// TIA Portal project "Street Light Control" (V17)
// Street Light Control
// The Street Light gets ON for 20s when there is any movement detected and then blinks with a interval of 1s, gets turned OFF after 30s.

(* hardware
DEVICE "S7-1200 station_1"  S7-1200 Station
   slot 0: "Rack_0"  S7-1200 Rack  Rack  V1.0
   slot 1: "PLC_1"  CPU 1215C DC/DC/DC  6ES7 215-1AG40-0XB0  V4.5
*)

// ===== PLC "PLC_1"  CPU 1215C DC/DC/DC =====

VAR_GLOBAL   // PLC tag table "Default tag table"
   "Motion_Sensor" AT %I0.1 : Bool;
   "Street_Lights" AT %Q0.0 : Bool;
   "Tag_1" AT %M0.0 : Bool;
   "Tag_2" AT %M0.1 : Bool;
   "Tag_3" AT %MD0 : Time;
   "Tag_4" AT %MD4 : Time;
   "PB" AT %I0.0 : Bool;
   "Tag_5" AT %M0.3 : Bool;
END_VAR

// folder: System blocks/Program resources

DATA_BLOCK "IEC_Timer_0_DB"   // DB1
{ S7_Optimized_Access := 'TRUE' }
AUTHOR : Simatic
FAMILY : IEC
NAME : IEC_TMR
VERSION : 1.0
// stored: InstanceOfName IEC_TIMER
"IEC_TIMER"
BEGIN
END_DATA_BLOCK

DATA_BLOCK "IEC_Timer_0_DB_1"   // DB2
{ S7_Optimized_Access := 'TRUE' }
AUTHOR : Simatic
FAMILY : IEC
NAME : IEC_TMR
VERSION : 1.0
// stored: InstanceOfName IEC_TIMER
"IEC_TIMER"
BEGIN
END_DATA_BLOCK

DATA_BLOCK "IEC_Timer_0_DB_2"   // DB3
{ S7_Optimized_Access := 'TRUE' }
AUTHOR : Simatic
FAMILY : IEC
NAME : IEC_TMR
VERSION : 1.0
// stored: InstanceOfName IEC_TIMER
"IEC_TIMER"
BEGIN
END_DATA_BLOCK

DATA_BLOCK "IEC_Timer_0_DB_4"   // DB5
{ S7_Optimized_Access := 'TRUE' }
AUTHOR : Simatic
FAMILY : IEC
NAME : IEC_TMR
VERSION : 1.0
// stored: InstanceOfName IEC_TIMER
"IEC_TIMER"
BEGIN
END_DATA_BLOCK

// folder: (top level)

ORGANIZATION_BLOCK "Main"   // OB1, LAD, ProgramCycle
TITLE = "Main Program Sweep (Cycle)"
{ S7_Optimized_Access := 'TRUE' }
VERSION : 0.1
   VAR_INPUT
      Initial_Call : Bool;   // Initial call of this OB
      Remanence : Bool;   // =True, if remanent data are available
   END_VAR
   VAR_TEMP   // added for the SCL form of the ladder/FBD networks
      _w1 : Bool;
   END_VAR
BEGIN

REGION Network 1
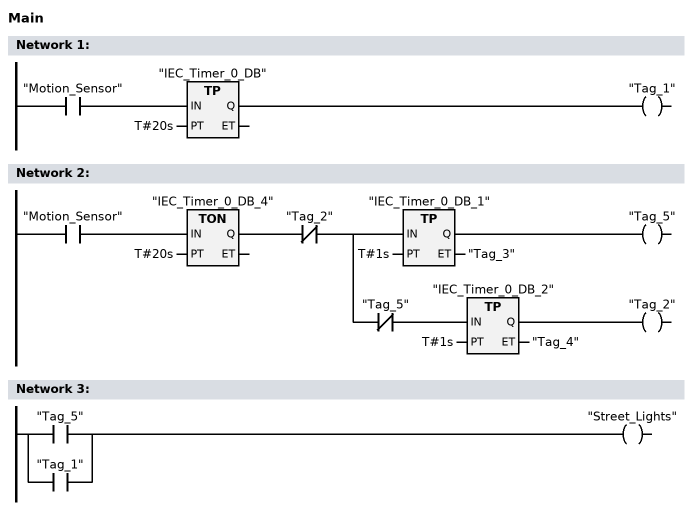
   "IEC_Timer_0_DB".TP(IN := "Motion_Sensor", PT := T#20s);
   "Tag_1" := "IEC_Timer_0_DB".Q;
END_REGION

REGION Network 2
   "IEC_Timer_0_DB_4".TON(IN := "Motion_Sensor", PT := T#20s);
   #_w1 := "IEC_Timer_0_DB_4".Q AND NOT "Tag_2";
   "IEC_Timer_0_DB_1".TP(IN := #_w1, PT := T#1s, ET => "Tag_3");
   "Tag_5" := "IEC_Timer_0_DB_1".Q;
   "IEC_Timer_0_DB_2".TP(IN := #_w1 AND NOT "Tag_5", PT := T#1s, ET => "Tag_4");
   "Tag_2" := "IEC_Timer_0_DB_2".Q;
END_REGION

REGION Network 3
   RUNG wire#powerrail
      Contact( "Tag_5" )
      wire#w1
      Coil( "Street_Lights" )
   END_RUNG
   RUNG wire#powerrail
      Contact( "Tag_1" )
   END_RUNG wire#w1
   // the same network as SCL:
   "Street_Lights" := "Tag_5" OR "Tag_1";
END_REGION
END_ORGANIZATION_BLOCK